// TwinCAT 3 PLC project PLC
// ProgramVersion: 3.1.4023.0
// libraries:
//   Tc2_MC2, * (Beckhoff Automation GmbH)
//   Tc2_PlcInterpolation, * (Beckhoff Automation GmbH)
//   Tc2_Standard, * (Beckhoff Automation GmbH)
//   Tc2_System, * (Beckhoff Automation GmbH)
//   Tc3_Module, * (Beckhoff Automation GmbH)
// project tree:
//   DUTs/ CASE_MODE.TcDUT, CASE_STATE.TcDUT, INIT_GVL.TcGVL, McOutputs.TcGVL, NCI_SingleEntry.TcDUT, PLCStruct.TcDUT, POS_REQ.TcDUT, POS_REQ_Resample.TcDUT, POS_RSP.TcDUT, POWER_GVL.TcGVL, RESET_GVL.TcGVL, TEST_STATE.TcDUT, VEL_REQ.TcDUT, VEL_RSP.TcDUT
//   / PlcTask.TcTTO
//   POUs/ AXIS.TcPOU, INIT.TcPOU, MAIN.TcPOU, Move_Vel.TcPOU, NCI_REF.TcPOU, POWER.TcPOU, PRG_MC_FeedTable.TcPOU, READ_POS.TcPOU, READ_VEL.TcPOU, RESET.TcPOU, SetPointGeneration.TcPOU, set_pos.TcPOU, TEST.TcPOU, TimeGet.TcPOU, WAIT.TcPOU

CONFIGURATION PLC
    RESOURCE PLC ON TwinCAT3
        TASK PlcTask(INTERVAL := T#50000us, PRIORITY := 20);
        PROGRAM MAIN WITH PlcTask : MAIN;
    END_RESOURCE
END_CONFIGURATION

// ---- DUTs/CASE_MODE.TcDUT

TYPE CASE_MODE :
(
	DEFAULT := 0,
	Set_PointGeneration,
	Set_Vel
);
END_TYPE

// ---- DUTs/CASE_STATE.TcDUT

TYPE CASE_STATE :
(
	ENUM_INIT_0 :=0,
	ENUM_POWER,
	ENUM_INIT,
	ENUM_SET_POSITION_GENERATION,
	ENUM_ERROR,
	ENUM_RESET
)INT;
END_TYPE

// ---- DUTs/NCI_SingleEntry.TcDUT
TYPE NCI_SingleEntry :
STRUCT
	SyncVelo:REAL;
	SyncAcc:REAL;
	fX:REAL;
	fY:REAL;
	fZ:REAL;
	
	fQ1:REAL;
	fQ2:REAL;
	
	fCenterX:REAL;
	fCenterY:REAL;
	fCenterZ:REAL;
	iPlane:REAL;
	
	Reserve1:UDINT;
	Reserve2:UDINT;
END_STRUCT
END_TYPE

// ---- DUTs/PLCStruct.TcDUT
TYPE PLCStruct :
STRUCT
	FLOAT1 :LREAL;
	FLOAT2 :LREAL;
	FLOAT3 :LREAL;
	FLOAT4 :LREAL;
(*
	intVal : INT;
	floatVal : REAL;
	boolVal : BOOL;
	*)
END_STRUCT
END_TYPE

// ---- DUTs/POS_REQ.TcDUT
TYPE POS_REQ :
STRUCT
	POS1: LREAL;
	POS2: LREAL;
	POS3: LREAL;
	POS4: LREAL;
	POS5: LREAL;
	POS6: LREAL;
END_STRUCT
END_TYPE

// ---- DUTs/POS_REQ_Resample.TcDUT
TYPE POS_REQ_Resample :
STRUCT
	POS_Resample: ARRAY[1..8,1..15] OF LREAL;
	(*POS1: LREAL;
	POS2: LREAL;
	POS3: LREAL;
	POS4: LREAL;
	POS5: LREAL;
	POS6: LREAL;*)

END_STRUCT
END_TYPE

// ---- DUTs/POS_RSP.TcDUT
TYPE POS_RSP :
STRUCT
	POS1: LREAL;
	POS2: LREAL;
	POS3: LREAL;
	POS4: LREAL;
	POS5: LREAL;
	POS6: LREAL;
END_STRUCT
END_TYPE

// ---- DUTs/TEST_STATE.TcDUT
TYPE TEST_STATE :
(
	TEST_0 :=0,
	TEST_1,
	TEST_2,
	TEST_3
)INT;
END_TYPE

// ---- DUTs/VEL_REQ.TcDUT
TYPE VEL_REQ :
STRUCT
	VEL5: LREAL;
	VEL6: LREAL;
END_STRUCT
END_TYPE

// ---- DUTs/VEL_RSP.TcDUT
TYPE VEL_RSP :
STRUCT
	VEL1: LREAL;
	VEL2: LREAL;
	VEL3: LREAL;
	VEL4: LREAL;
	VEL5: LREAL;
	VEL6: LREAL;
END_STRUCT
END_TYPE

// ---- DUTs/INIT_GVL.TcGVL

VAR_GLOBAL
	INIT_Execute1 : BOOL;
	INIT_Execute2 : BOOL;
	INIT_Execute3 : BOOL;
	INIT_Execute4 : BOOL;
	INIT_Execute5 : BOOL;
	INIT_Execute6 : BOOL;
END_VAR

// ---- DUTs/McOutputs.TcGVL

VAR_GLOBAL
	MC_Power_Outputs1: ST_McOutputs;
	MC_Power_Outputs2: ST_McOutputs;
	MC_Power_Outputs3: ST_McOutputs;
	MC_Power_Outputs4: ST_McOutputs;
	MC_Power_Outputs5: ST_McOutputs;
	MC_Power_Outputs6: ST_McOutputs;
END_VAR

// ---- DUTs/POWER_GVL.TcGVL

VAR_GLOBAL
	POWER_Enable1 : BOOL;
	POWER_Enable2 : BOOL;
	POWER_Enable3 : BOOL;
	POWER_Enable4 : BOOL;
	POWER_Enable5 : BOOL;
	POWER_Enable6 : BOOL;
END_VAR

// ---- DUTs/RESET_GVL.TcGVL

VAR_GLOBAL
	RESET_Execute1 : BOOL;
	RESET_Execute2 : BOOL;
	RESET_Execute3 : BOOL;
	RESET_Execute4 : BOOL;
	RESET_Execute5 : BOOL;
	RESET_Execute6 : BOOL;
END_VAR

// ---- POUs/MAIN.TcPOU
PROGRAM MAIN
VAR
	//BOOL1 AT %MX0.0 :BOOL;
	//INT2 AT %MD2 :INT;
	//FLOAT1 AT %MD6:REAL;
	//String1 : STRING;
	//Array1 : ARRAY[0..9] OF INT;
	//PLCVar:PLCStruct;
	//ArrayS:ARRAY[0..9] OF PLCStruct;
	//array2: ARRAY[1..50] OF LREAL:=[1,2,3,4,5,6,7,8,9,10,11,12,13,14,15,16,17,18,19,20,21,22,23,24,25,26,27,28,29,30,31,32,33,34,35,36,37,38,39,40,41,42,43,44,45,46,47,48,49,50];
	//TON1: TON;	
	//count: INT;
	//CTU1: CTU;

	CASE_MODE1 :CASE_MODE;
	FillFlag AT %MX0.0: BOOL;
	MoveDoneFlag AT %MX1.0: BOOL;
	Move_Stop_Flag AT %MX2.0: BOOL;
	Power_Flag AT %MX3.0: BOOL;
	Init_Flag AT %MX12.0: BOOL;
	NoPower_Flag AT %MX5.0: BOOL;
	Reset_Flag AT %MX6.0: BOOL;
	Continue_Flag AT %MX7.0: BOOL;
	Mode_Flag AT %MD8: INT;
	test1 AT %MX10.0: BOOL;
	test2 AT %MX11.0: BOOL;
	start_flag AT %MX9.0: BOOL;
	set_pos_flag AT %MX13.0: BOOL;
	err_flag AT %MX14.0: BOOL;
	Init_Done_flag AT %MX15.0: BOOL;
	MovePermit_Flag: BOOL;
	POS1_temp: LREAL;
	POS2_temp: LREAL;
	POS3_temp: LREAL;
	POS4_temp: LREAL;
	Done1Flag: LREAL;
	Done2Flag: LREAL;
	Done3Flag: LREAL;
	Done4Flag: LREAL;
	i: INT;
	x AT %MW2: INT;
	POS_REQ :POS_REQ;
	POS_RSP1 :POS_RSP;
	VEL_RSP1 :VEL_RSP;
	POS_REQ_Resample1:POS_REQ_Resample;	
	VEL_REQ1 :VEL_REQ;
	
	j: INT;
	m: INT;
	fbGetCurTaskIdx  : GETCURTASKINDEX;
    nLastExecTime       : UDINT;
	init_done_1: BOOL;
	init_done_2: BOOL;
	init_done_3: BOOL;
	init_done_4: BOOL;
	init_done_5: BOOL;
	init_done_6: BOOL;
END_VAR

//PRG_MC_FeedTable();
AXIS();
READ_POS();
READ_VEL();
//	IF AXIS.axis1.Status.Error AND AXIS.axis2.Status.Error AND AXIS.axis3.Status.Error AND AXIS.axis4.Status.Error THEN
//		start_flag:=0;
//	ELSE
//		start_flag:=1;
//	END_IF

		IF 	Move_Stop_Flag THEN
			MovePermit_Flag :=FALSE;
		END_IF
		IF Continue_Flag AND NOT err_flag THEN
			Move_Stop_Flag:= 0;
			MovePermit_Flag :=TRUE;
			Continue_Flag:= 0;
		END_IF
		IF Init_Flag AND NOT err_flag THEN
			POWER_Enable1:=TRUE; 
			POWER_Enable2:=TRUE;
			POWER_Enable3:=TRUE;
			POWER_Enable4:=TRUE;
			POWER();
			IF MC_Power_Outputs1.Done  AND MC_Power_Outputs2.Done AND MC_Power_Outputs3.Done AND MC_Power_Outputs4.Done THEN
				Power_Flag:= TRUE;
				INIT.MC_MoveAbsolute_1(Axis:=AXIS.Axis1,Execute:=TRUE,Position:=0,Velocity:=300);
				INIT.MC_MoveAbsolute_2(Axis:=AXIS.Axis2,Execute:=TRUE,Position:=0,Velocity:=300);
				INIT.MC_MoveAbsolute_3(Axis:=AXIS.Axis3,Execute:=TRUE,Position:=0,Velocity:=300);
				INIT.MC_MoveAbsolute_4(Axis:=AXIS.Axis4,Execute:=TRUE,Position:=0,Velocity:=300);
				IF NOT INIT.MC_MoveAbsolute_1.busy THEN
					init_done_1 := TRUE;
				END_IF
				IF NOT INIT.MC_MoveAbsolute_2.busy THEN
					init_done_2 := TRUE;
				END_IF
				IF NOT INIT.MC_MoveAbsolute_3.busy THEN
					init_done_3 := TRUE;
				END_IF
				IF NOT INIT.MC_MoveAbsolute_4.busy THEN
					init_done_4 := TRUE;
				END_IF
				IF init_done_1 AND init_done_2 AND init_done_3 AND init_done_4 THEN
					INIT.MC_MoveAbsolute_1(Axis:=AXIS.Axis1,Execute:=FALSE);
					INIT.MC_MoveAbsolute_2(Axis:=AXIS.Axis2,Execute:=FALSE);
					INIT.MC_MoveAbsolute_3(Axis:=AXIS.Axis3,Execute:=FALSE);
					INIT.MC_MoveAbsolute_4(Axis:=AXIS.Axis4,Execute:=FALSE);
					init_done_1 :=FALSE;
					init_done_2 :=FALSE;
					init_done_3 :=FALSE;
					init_done_4 :=FALSE;
					SetPointGeneration.MC_ExtSetPointGenEnable1(Axis:=AXIS.Axis1,Execute:=FALSE);	
					SetPointGeneration.MC_ExtSetPointGenEnable2(Axis:=AXIS.Axis2,Execute:=FALSE);
					SetPointGeneration.MC_ExtSetPointGenEnable3(Axis:=AXIS.Axis3,Execute:=FALSE);
					SetPointGeneration.MC_ExtSetPointGenEnable4(Axis:=AXIS.Axis4,Execute:=FALSE);
					SetPointGeneration.MC_ExtSetPointGenDisable1(Axis:=AXIS.Axis1,Execute:=FALSE);	
					SetPointGeneration.MC_ExtSetPointGenDisable2(Axis:=AXIS.Axis2,Execute:=FALSE);
					SetPointGeneration.MC_ExtSetPointGenDisable3(Axis:=AXIS.Axis3,Execute:=FALSE);
					SetPointGeneration.MC_ExtSetPointGenDisable4(Axis:=AXIS.Axis4,Execute:=FALSE);
					Init_Flag:= 0;
					Power_Flag:= 0;
					MovePermit_Flag:= 1;
					Init_Done_flag:=1;
				END_IF
			END_IF
			IF AXIS.axis1.Status.Error AND AXIS.axis2.Status.Error AND AXIS.axis3.Status.Error AND AXIS.axis4.Status.Error THEN
				err_flag:=1;
			END_IF					
		END_IF
		
		IF set_pos_flag THEN
			set_pos.MC_SetPosition1(axis:=axis.Axis1,execute:=FALSE,position:=0);
			set_pos.MC_SetPosition2(axis:=axis.Axis2,execute:=FALSE,position:=0);
			set_pos.MC_SetPosition3(axis:=axis.Axis3,execute:=FALSE,position:=0);
			set_pos.MC_SetPosition4(axis:=axis.Axis4,execute:=FALSE,position:=0);
			set_pos.MC_SetPosition1(axis:=axis.Axis1,execute:=TRUE,position:=0);
			set_pos.MC_SetPosition2(axis:=axis.Axis2,execute:=TRUE,position:=0);
			set_pos.MC_SetPosition3(axis:=axis.Axis3,execute:=TRUE,position:=0);
			set_pos.MC_SetPosition4(axis:=axis.Axis4,execute:=TRUE,position:=0);
			set_pos_flag:=0;
		END_IF
		
		IF Reset_Flag THEN
			SetPointGeneration.MC_ExtSetPointGenDisable1(Axis:=AXIS.Axis1,Execute:=TRUE);	
			SetPointGeneration.MC_ExtSetPointGenDisable2(Axis:=AXIS.Axis2,Execute:=TRUE);
			SetPointGeneration.MC_ExtSetPointGenDisable3(Axis:=AXIS.Axis3,Execute:=TRUE);
			SetPointGeneration.MC_ExtSetPointGenDisable4(Axis:=AXIS.Axis4,Execute:=TRUE);
			INIT.MC_MoveAbsolute_1(Axis:=AXIS.Axis1,Execute:=FALSE);
			INIT.MC_MoveAbsolute_2(Axis:=AXIS.Axis2,Execute:=FALSE);
			INIT.MC_MoveAbsolute_3(Axis:=AXIS.Axis3,Execute:=FALSE);
			INIT.MC_MoveAbsolute_4(Axis:=AXIS.Axis4,Execute:=FALSE);
			Init_Flag :=FALSE;
			POWER_Enable1:=FALSE;
			POWER_Enable2:=FALSE;
			POWER_Enable3:=FALSE;
			POWER_Enable4:=FALSE;
			POWER();
			Power_Flag :=0;
			RESET.MC_Reset1(Axis:=AXIS.Axis1,Execute:=TRUE);
			RESET.MC_Reset2(Axis:=AXIS.Axis2,Execute:=TRUE);
			RESET.MC_Reset3(Axis:=AXIS.Axis3,Execute:=TRUE);
			RESET.MC_Reset4(Axis:=AXIS.Axis4,Execute:=TRUE);
			RESET.MC_Reset1(Axis:=AXIS.Axis1,Execute:=FALSE);
			RESET.MC_Reset2(Axis:=AXIS.Axis2,Execute:=FALSE);
			RESET.MC_Reset3(Axis:=AXIS.Axis3,Execute:=FALSE);
			RESET.MC_Reset4(Axis:=AXIS.Axis4,Execute:=FALSE);
			Reset_Flag:= 0;
			Init_Done_flag:=0;
			NoPower_Flag:= 0;
			Move_Stop_Flag:= 0;
			MovePermit_Flag:= 0;
			start_flag:=0;
		END_IF
		IF NoPower_Flag AND NOT err_flag THEN
			MovePermit_Flag:= 0;
			Init_Flag:= 0;
			NoPower_Flag:= FALSE;
			POWER_Enable1:=FALSE;
			POWER_Enable2:=FALSE;
			POWER_Enable3:=FALSE;
			POWER_Enable4:=FALSE;
			POWER();
	//IF SetPointGeneration.MC_Power_1_Outputs.Done AND SetPointGeneration.MC_Power_2_Outputs.Done AND SetPointGeneration.MC_Power_3_Outputs.Done AND SetPointGeneration.MC_Power_4_Outputs.Done THEN
		
	//END_IF	
		END_IF
		IF MovePermit_Flag AND NOT err_flag THEN
			FillFlag:= FALSE;
			IF MOve_Stop_Flag THEN
				;
			ELSE
				i:= i+1;
			END_IF

			x:= i MOD 15;
	
			POS_RSP1.POS1:= AXIS.Axis1.NcToPlc.actPos;
			POS_RSP1.POS2:= AXIS.Axis2.NcToPlc.actPos;
			POS_RSP1.POS3:= AXIS.Axis3.NcToPlc.actPos;
			POS_RSP1.POS4:= AXIS.Axis4.NcToPlc.actPos;
			VEL_RSP1.VEL1:= AXIS.Axis1.NcToPlc.actVelo;
			VEL_RSP1.VEL2:= AXIS.Axis2.NcToPlc.actVelo;
			VEL_RSP1.VEL3:= AXIS.Axis3.NcToPlc.actVelo;
			VEL_RSP1.VEL4:= AXIS.Axis4.NcToPlc.actVelo;
			Done1Flag:=AXIS.Axis1.NcToPlc.actPos-POS1_temp;
			Done2Flag:=AXIS.Axis2.NcToPlc.actPos-POS2_temp;
			Done3Flag:=AXIS.Axis3.NcToPlc.actPos-POS3_temp;
			Done4Flag:=AXIS.Axis4.NcToPlc.actPos-POS4_temp;

			IF MOve_Stop_Flag = 0 AND ABS(Done1Flag)<1E-3 AND ABS(Done2Flag)<1E-3 AND ABS(Done3Flag)<1E-3 AND ABS(Done4Flag)<1E-3 THEN
				MoveDoneFlag:= 1;
			ELSE
				MoveDoneFlag:= 0;
			END_IF
	
			POS_REQ.POS1:= -POS_REQ_Resample1.POS_Resample[3,x+1];
			POS_REQ.POS2:= -POS_REQ_Resample1.POS_Resample[4,x+1];
			POS_REQ.POS3:= -POS_REQ_Resample1.POS_Resample[1,x+1];
			POS_REQ.POS4:= -POS_REQ_Resample1.POS_Resample[2,x+1];
			IF POS_REQ_Resample1.POS_Resample[7,x] = 1 THEN
				POS1_temp:= POS_REQ.POS1;
			END_IF
			IF POS_REQ_Resample1.POS_Resample[8,x] = 1 THEN
				POS2_temp:= POS_REQ.POS2;
			END_IF
			IF POS_REQ_Resample1.POS_Resample[5,x] = 1 THEN
				POS3_temp:= POS_REQ.POS3;
			END_IF
			IF POS_REQ_Resample1.POS_Resample[6,x] = 1 THEN
				POS4_temp:= POS_REQ.POS4;
			END_IF

		SetPointGeneration.MC_ExtSetPointGenEnable1(Axis:=AXIS.Axis1,Execute:=TRUE,Position:=POS_REQ.POS1);	
		SetPointGeneration.MC_ExtSetPointGenEnable2(Axis:=AXIS.Axis2,Execute:=TRUE,Position:=POS_REQ.POS2);
		SetPointGeneration.MC_ExtSetPointGenEnable3(Axis:=AXIS.Axis3,Execute:=TRUE,Position:=POS_REQ.POS3);
		SetPointGeneration.MC_ExtSetPointGenEnable4(Axis:=AXIS.Axis4,Execute:=TRUE,Position:=POS_REQ.POS4);
		IF SetPointGeneration.MC_ExtSetPointGenEnable1.Enabled AND  SetPointGeneration.MC_ExtSetPointGenEnable2.Enabled AND  SetPointGeneration.MC_ExtSetPointGenEnable3.Enabled AND  SetPointGeneration.MC_ExtSetPointGenEnable4.Enabled THEN
			MC_ExtSetPointGenFeed(
				Position:= MAIN.POS_REQ.POS1, 		
				Velocity:= 1, 
				Acceleration:=1 , 
				Direction:= 1,
				Axis:= AXIS.Axis1);	
			MC_ExtSetPointGenFeed(
				Position:= MAIN.POS_REQ.POS2, 		
				Velocity:= 1, 
				Acceleration:=1 , 
				Direction:= 1,
				Axis:= AXIS.Axis2);	
			MC_ExtSetPointGenFeed(
				Position:= MAIN.POS_REQ.POS3, 		
				Velocity:= 1, 
				Acceleration:=1 , 
				Direction:= 1,
				Axis:= AXIS.Axis3);	
			MC_ExtSetPointGenFeed(
				Position:= MAIN.POS_REQ.POS4, 		
				Velocity:= 1, 
				Acceleration:=1 , 
				Direction:= 1,
				Axis:= AXIS.Axis4);		
				
		END_IF
		IF AXIS.axis1.Status.Error AND AXIS.axis2.Status.Error AND AXIS.axis3.Status.Error AND AXIS.axis4.Status.Error THEN
			err_flag := 1;
		END_IF
	
			IF x = 14 AND MOve_Stop_Flag = 0 THEN
				FillFlag:= TRUE;
		(*FOR m:= 1 TO 15 DO
			POS_REQ_Resample1.POS_Resample[1,m]:=15*j+m;
		END_FOR
		j:= j+1;*)
			END_IF
	
		END_IF
		IF err_flag THEN
			Reset_Flag:=1;
			IF NOT AXIS.axis1.Status.Error AND NOT AXIS.axis2.Status.Error AND NOT AXIS.axis3.Status.Error AND NOT AXIS.axis4.Status.Error THEN
				err_flag := 0;
			END_IF
		END_IF
		
fbGetCurTaskIdx();
nLastExecTime := _TaskInfo[fbGetCurTaskIdx.index].LastExecTime;

END_PROGRAM

// ---- POUs/AXIS.TcPOU
PROGRAM AXIS
VAR
	Axis1: AXIS_REF;
	Axis2: AXIS_REF;
	Axis3: AXIS_REF;
	Axis4: AXIS_REF;
	Axis5: AXIS_REF;
	Axis6: AXIS_REF;
END_VAR

Axis1(
	PlcToNc:= , 
	NcToPlc=> , 
	ADS=> , 
	Status=> , 
	DriveAddress:= );
	
Axis2(
	PlcToNc:= , 
	NcToPlc=> , 
	ADS=> , 
	Status=> , 
	DriveAddress:= );
	
Axis3(
	PlcToNc:= , 
	NcToPlc=> , 
	ADS=> , 
	Status=> , 
	DriveAddress:= );
	
Axis4(
	PlcToNc:= , 
	NcToPlc=> , 
	ADS=> , 
	Status=> , 
	DriveAddress:= );

Axis5(
	PlcToNc:= , 
	NcToPlc=> , 
	ADS=> , 
	Status=> , 
	DriveAddress:= );
	
Axis6(
	PlcToNc:= , 
	NcToPlc=> , 
	ADS=> , 
	Status=> , 
	DriveAddress:= );

END_PROGRAM

// ---- POUs/READ_POS.TcPOU
PROGRAM READ_POS
VAR
	MC_ReadActualPosition1 : MC_ReadActualPosition;
	MC_ReadActualPosition2 : MC_ReadActualPosition;
	MC_ReadActualPosition3 : MC_ReadActualPosition;
	MC_ReadActualPosition4 : MC_ReadActualPosition;
END_VAR

MC_ReadActualPosition1(
	Axis:= AXIS.Axis1, 
	Enable:= , 
	Valid=> , 
	Busy=> , 
	Error=> , 
	ErrorID=> , 
	Position=> );
	
MC_ReadActualPosition2(
	Axis:= AXIS.Axis2, 
	Enable:= , 
	Valid=> , 
	Busy=> , 
	Error=> , 
	ErrorID=> , 
	Position=> );
	
MC_ReadActualPosition3(
	Axis:= AXIS.Axis3, 
	Enable:= , 
	Valid=> , 
	Busy=> , 
	Error=> , 
	ErrorID=> , 
	Position=> );
	
MC_ReadActualPosition4(
	Axis:= AXIS.Axis4, 
	Enable:= , 
	Valid=> , 
	Busy=> , 
	Error=> , 
	ErrorID=> , 
	Position=> );

END_PROGRAM

// ---- POUs/READ_VEL.TcPOU
PROGRAM READ_VEL
VAR
	MC_ReadActualVelocity1 : MC_ReadActualVelocity;
	MC_ReadActualVelocity2 : MC_ReadActualVelocity;
	MC_ReadActualVelocity3 : MC_ReadActualVelocity;
	MC_ReadActualVelocity4 : MC_ReadActualVelocity;
END_VAR

MC_ReadActualVelocity1(
	Axis:= AXIS.Axis1, 
	Enable:= , 
	Valid=> , 
	Busy=> , 
	Error=> , 
	ErrorID=> , 
	ActualVelocity=> );
	
MC_ReadActualVelocity2(
	Axis:= AXIS.Axis2, 
	Enable:= , 
	Valid=> , 
	Busy=> , 
	Error=> , 
	ErrorID=> , 
	ActualVelocity=> );
	
MC_ReadActualVelocity3(
	Axis:= AXIS.Axis3, 
	Enable:= , 
	Valid=> , 
	Busy=> , 
	Error=> , 
	ErrorID=> , 
	ActualVelocity=> );
	
MC_ReadActualVelocity4(
	Axis:= AXIS.Axis4, 
	Enable:= , 
	Valid=> , 
	Busy=> , 
	Error=> , 
	ErrorID=> , 
	ActualVelocity=> );

END_PROGRAM

// ---- POUs/POWER.TcPOU
PROGRAM POWER
VAR
	MC_Power_1: MC_Power;
	MC_Power_2: MC_Power;
	MC_Power_3: MC_Power;
	MC_Power_4: MC_Power;
	MC_Power_5: MC_Power;
	MC_Power_6: MC_Power;
	
END_VAR

MC_Power_1(
	Axis:= AXIS.Axis1, 
	Enable:= POWER_Enable1, 
	Enable_Positive:= POWER_Enable1, 
	Enable_Negative:= POWER_Enable1, 
	Override:= , 
	BufferMode:= , 
	Options:= , 
	Status=> MC_Power_Outputs1.Done, 
	Busy=> MC_Power_Outputs1.Busy, 
	Active=> MC_Power_Outputs1.Active, 
	Error=> MC_Power_Outputs1.Error, 
	ErrorID=> MC_Power_Outputs1.ErrorID);
	
MC_Power_2(
	Axis:= AXIS.Axis2, 
	Enable:= POWER_Enable2, 
	Enable_Positive:= POWER_Enable2, 
	Enable_Negative:= POWER_Enable2, 
	Override:= , 
	BufferMode:= , 
	Options:= , 
	Status=> MC_Power_Outputs2.Done, 
	Busy=> MC_Power_Outputs2.Busy, 
	Active=> MC_Power_Outputs2.Active, 
	Error=> MC_Power_Outputs2.Error, 
	ErrorID=> MC_Power_Outputs2.ErrorID);
	
MC_Power_3(
	Axis:= AXIS.Axis3, 
	Enable:= POWER_Enable3, 
	Enable_Positive:= POWER_Enable3, 
	Enable_Negative:= POWER_Enable3, 
	Override:= , 
	BufferMode:= , 
	Options:= , 
	Status=> MC_Power_Outputs3.Done, 
	Busy=> MC_Power_Outputs3.Busy, 
	Active=> MC_Power_Outputs3.Active, 
	Error=> MC_Power_Outputs3.Error, 
	ErrorID=> MC_Power_Outputs3.ErrorID);
	
MC_Power_4(
	Axis:= AXIS.Axis4, 
	Enable:= POWER_Enable4, 
	Enable_Positive:= POWER_Enable4, 
	Enable_Negative:= POWER_Enable4, 
	Override:= , 
	BufferMode:= , 
	Options:= , 
	Status=> MC_Power_Outputs4.Done, 
	Busy=> MC_Power_Outputs4.Busy, 
	Active=> MC_Power_Outputs4.Active, 
	Error=> MC_Power_Outputs4.Error, 
	ErrorID=> MC_Power_Outputs4.ErrorID);
	
MC_Power_5(
	Axis:= AXIS.Axis5, 
	Enable:= POWER_Enable5, 
	Enable_Positive:= POWER_Enable5, 
	Enable_Negative:= POWER_Enable5, 
	Override:= , 
	BufferMode:= , 
	Options:= , 
	Status=> MC_Power_Outputs5.Done, 
	Busy=> MC_Power_Outputs5.Busy, 
	Active=> MC_Power_Outputs5.Active, 
	Error=> MC_Power_Outputs5.Error, 
	ErrorID=> MC_Power_Outputs5.ErrorID);
	
MC_Power_6(
	Axis:= AXIS.Axis6, 
	Enable:= POWER_Enable6, 
	Enable_Positive:= POWER_Enable6, 
	Enable_Negative:= POWER_Enable6, 
	Override:= , 
	BufferMode:= , 
	Options:= , 
	Status=> MC_Power_Outputs6.Done, 
	Busy=> MC_Power_Outputs6.Busy, 
	Active=> MC_Power_Outputs6.Active, 
	Error=> MC_Power_Outputs6.Error, 
	ErrorID=> MC_Power_Outputs6.ErrorID);

END_PROGRAM

// ---- POUs/INIT.TcPOU
PROGRAM INIT
VAR
	MC_MoveAbsolute_1 : MC_MoveAbsolute;
	MC_MoveAbsolute_2 : MC_MoveAbsolute;
	MC_MoveAbsolute_3 : MC_MoveAbsolute;
	MC_MoveAbsolute_4 : MC_MoveAbsolute;
	MC_MoveAbsolute_5 : MC_MoveAbsolute;
	MC_MoveAbsolute_6 : MC_MoveAbsolute;
END_VAR

MC_MoveAbsolute_1(
	Axis:= AXIS.Axis1, 
	Execute:= INIT_Execute1, 
	Position:= , 
	Velocity:= , 
	Acceleration:= , 
	Deceleration:= , 
	Jerk:= , 
	BufferMode:= , 
	Options:= , 
	Done=> , 
	Busy=> , 
	Active=> , 
	CommandAborted=> , 
	Error=> , 
	ErrorID=> );
	
MC_MoveAbsolute_2(
	Axis:= AXIS.Axis2, 
	Execute:= INIT_Execute2, 
	Position:= , 
	Velocity:= , 
	Acceleration:= , 
	Deceleration:= , 
	Jerk:= , 
	BufferMode:= , 
	Options:= , 
	Done=> , 
	Busy=> , 
	Active=> , 
	CommandAborted=> , 
	Error=> , 
	ErrorID=> );
	
MC_MoveAbsolute_3(
	Axis:= AXIS.Axis3, 
	Execute:= INIT_Execute3, 
	Position:= , 
	Velocity:= , 
	Acceleration:= , 
	Deceleration:= , 
	Jerk:= , 
	BufferMode:= , 
	Options:= , 
	Done=> , 
	Busy=> , 
	Active=> , 
	CommandAborted=> , 
	Error=> , 
	ErrorID=> );
	
MC_MoveAbsolute_4(
	Axis:= AXIS.Axis4, 
	Execute:= INIT_Execute4, 
	Position:= , 
	Velocity:= , 
	Acceleration:= , 
	Deceleration:= , 
	Jerk:= , 
	BufferMode:= , 
	Options:= , 
	Done=> , 
	Busy=> , 
	Active=> , 
	CommandAborted=> , 
	Error=> , 
	ErrorID=> );
	
MC_MoveAbsolute_5(
	Axis:= AXIS.Axis5, 
	Execute:= INIT_Execute5, 
	Position:= , 
	Velocity:= , 
	Acceleration:= , 
	Deceleration:= , 
	Jerk:= , 
	BufferMode:= , 
	Options:= , 
	Done=> , 
	Busy=> , 
	Active=> , 
	CommandAborted=> , 
	Error=> , 
	ErrorID=> );
	
MC_MoveAbsolute_6(
	Axis:= AXIS.Axis6, 
	Execute:= INIT_Execute6, 
	Position:= , 
	Velocity:= , 
	Acceleration:= , 
	Deceleration:= , 
	Jerk:= , 
	BufferMode:= , 
	Options:= , 
	Done=> , 
	Busy=> , 
	Active=> , 
	CommandAborted=> , 
	Error=> , 
	ErrorID=> );

END_PROGRAM

// ---- POUs/SetPointGeneration.TcPOU
PROGRAM SetPointGeneration
VAR
	
	CASE_STATE1: CASE_STATE;
	
	MC_ExtSetPointGenEnable1: MC_ExtSetPointGenEnable;
	MC_ExtSetPointGenEnable2: MC_ExtSetPointGenEnable;
	MC_ExtSetPointGenEnable3: MC_ExtSetPointGenEnable;
	MC_ExtSetPointGenEnable4: MC_ExtSetPointGenEnable;
	
	MC_ExtSetPointGenDisable1: MC_ExtSetPointGenDisable;
	MC_ExtSetPointGenDisable2: MC_ExtSetPointGenDisable;
	MC_ExtSetPointGenDisable3: MC_ExtSetPointGenDisable;
	MC_ExtSetPointGenDisable4: MC_ExtSetPointGenDisable;
	
END_VAR

AXIS();



MC_ExtSetPointGenEnable1(
	Axis:= AXIS.Axis1, 
	Execute:= , 
	Position:= , 
	PositionType:= , 
	Done=> , 
	Busy=> , 
	Error=> , 
	ErrorID=> , 
	Enabled=> );
	
MC_ExtSetPointGenEnable2(
	Axis:= AXIS.Axis2, 
	Execute:= , 
	Position:= , 
	PositionType:= , 
	Done=> , 
	Busy=> , 
	Error=> , 
	ErrorID=> , 
	Enabled=> );
	
MC_ExtSetPointGenEnable3(
	Axis:= AXIS.Axis3, 
	Execute:= , 
	Position:= , 
	PositionType:= , 
	Done=> , 
	Busy=> , 
	Error=> , 
	ErrorID=> , 
	Enabled=> );
	
MC_ExtSetPointGenEnable4(
	Axis:= AXIS.Axis4, 
	Execute:= , 
	Position:= , 
	PositionType:= , 
	Done=> , 
	Busy=> , 
	Error=> , 
	ErrorID=> , 
	Enabled=> );
	
	MC_ExtSetPointGenDisable1(
	Axis:= AXIS.Axis1, 
	Execute:= , 
	Done=> , 
	Busy=> , 
	Error=> , 
	ErrorID=> , 
	Enabled=> );
	
	MC_ExtSetPointGenDisable2(
	Axis:= AXIS.Axis2, 
	Execute:= , 
	Done=> , 
	Busy=> , 
	Error=> , 
	ErrorID=> , 
	Enabled=> );
	
	MC_ExtSetPointGenDisable3(
	Axis:= AXIS.Axis3, 
	Execute:= , 
	Done=> , 
	Busy=> , 
	Error=> , 
	ErrorID=> , 
	Enabled=> );
	
	MC_ExtSetPointGenDisable4(
	Axis:= AXIS.Axis4, 
	Execute:= , 
	Done=> , 
	Busy=> , 
	Error=> , 
	ErrorID=> , 
	Enabled=> );

	
		
	
//	ENUM_ERROR:
//		MC_ExtSetPointGenEnable1.Execute:=FALSE;
//		MC_ExtSetPointGenEnable2.Execute:=FALSE;
//		MC_ExtSetPointGenEnable3.Execute:=FALSE;
//		MC_ExtSetPointGenEnable4.Execute:=FALSE;
//		MC_ExtSetPointGenDisable1.Execute := MC_ExtSetPointGenEnable1.Enabled;	
//		MC_ExtSetPointGenDisable2.Execute := MC_ExtSetPointGenEnable2.Enabled;
//		MC_ExtSetPointGenDisable3.Execute := MC_ExtSetPointGenEnable3.Enabled;
//		MC_ExtSetPointGenDisable4.Execute := MC_ExtSetPointGenEnable4.Enabled;	
//		IF NOT AXIS.axis1.Status.Coupled AND AXIS.axis2.Status.Coupled AND AXIS.axis3.Status.Coupled AND AXIS.axis4.Status.Coupled THEN
//			IF AXIS.axis1.Status.Error AND AXIS.axis2.Status.Error AND AXIS.axis3.Status.Error AND AXIS.axis4.Status.Error THEN
//				CASE_STATE1 := ENUM_RESET;	
//			ELSE
//				CASE_STATE1 := ENUM_INIT_0;
//			END_IF
//		END_IF
	
//	ENUM_RESET:
//		RESET_Execute1 := TRUE;
//		RESET_Execute2 := TRUE;
//		RESET_Execute3 := TRUE;
//		RESET_Execute4 := TRUE;
//		RESET();
//		MC_ExtSetPointGenDisable1.Execute:=FALSE;
//		MC_ExtSetPointGenDisable2.Execute:=FALSE;
//		MC_ExtSetPointGenDisable3.Execute:=FALSE;
//		MC_ExtSetPointGenDisable4.Execute:=FALSE;		
//			IF RESET.MC_Reset1.Done AND RESET.MC_Reset2.Done AND RESET.MC_Reset3.Done AND RESET.MC_Reset4.Done THEN
//				CASE_STATE1 := ENUM_INIT_0;
//			ELSIF RESET.MC_Reset1.Error AND RESET.MC_Reset2.Error AND RESET.MC_Reset3.Error AND RESET.MC_Reset4.Error THEN
//				CASE_STATE1 := ENUM_INIT_0; 
//			END_IF

END_PROGRAM

// ---- POUs/set_pos.TcPOU
PROGRAM set_pos
VAR
	MC_SetPosition1: MC_SetPosition;
	MC_SetPosition2: MC_SetPosition;
	MC_SetPosition3: MC_SetPosition;
	MC_SetPosition4: MC_SetPosition;
	MC_SetPosition5: MC_SetPosition;
	MC_SetPosition6: MC_SetPosition;
END_VAR

MC_SetPosition1(
	Axis:= axis.Axis1, 
	Execute:= , 
	Position:= , 
	Mode:= , 
	Options:= , 
	Done=> , 
	Busy=> , 
	Error=> , 
	ErrorID=> );

MC_SetPosition2(
	Axis:= axis.Axis2, 
	Execute:= , 
	Position:= , 
	Mode:= , 
	Options:= , 
	Done=> , 
	Busy=> , 
	Error=> , 
	ErrorID=> );
	
MC_SetPosition3(
	Axis:= axis.Axis3, 
	Execute:= , 
	Position:= , 
	Mode:= , 
	Options:= , 
	Done=> , 
	Busy=> , 
	Error=> , 
	ErrorID=> );

MC_SetPosition4(
	Axis:= axis.Axis4, 
	Execute:= , 
	Position:= , 
	Mode:= , 
	Options:= , 
	Done=> , 
	Busy=> , 
	Error=> , 
	ErrorID=> );
	
MC_SetPosition5(
	Axis:= axis.Axis5, 
	Execute:= , 
	Position:= , 
	Mode:= , 
	Options:= , 
	Done=> , 
	Busy=> , 
	Error=> , 
	ErrorID=> );

MC_SetPosition6(
	Axis:= axis.Axis6, 
	Execute:= , 
	Position:= , 
	Mode:= , 
	Options:= , 
	Done=> , 
	Busy=> , 
	Error=> , 
	ErrorID=> );

END_PROGRAM

// ---- POUs/RESET.TcPOU
PROGRAM RESET
VAR
	MC_Reset1 : MC_Reset;
	MC_Reset2 : MC_Reset;
	MC_Reset3 : MC_Reset;
	MC_Reset4 : MC_Reset;
	MC_Reset5 : MC_Reset;
	MC_Reset6 : MC_Reset;
END_VAR

MC_Reset1(
	Axis:= AXIS.Axis1, 
	Execute:= RESET_Execute1, 
	Done=> , 
	Busy=> , 
	Error=> , 
	ErrorID=> );
	
	MC_Reset2(
	Axis:= AXIS.Axis2, 
	Execute:= RESET_Execute2, 
	Done=> , 
	Busy=> , 
	Error=> , 
	ErrorID=> );
	
	MC_Reset3(
	Axis:= AXIS.Axis3, 
	Execute:= RESET_Execute3, 
	Done=> , 
	Busy=> , 
	Error=> , 
	ErrorID=> );
	
	MC_Reset4(
	Axis:= AXIS.Axis4, 
	Execute:= RESET_Execute4, 
	Done=> , 
	Busy=> , 
	Error=> , 
	ErrorID=> );
	
	MC_Reset5(
	Axis:= AXIS.Axis5, 
	Execute:= RESET_Execute5, 
	Done=> , 
	Busy=> , 
	Error=> , 
	ErrorID=> );
	
	MC_Reset6(
	Axis:= AXIS.Axis6, 
	Execute:= RESET_Execute6, 
	Done=> , 
	Busy=> , 
	Error=> , 
	ErrorID=> );

END_PROGRAM

// ---- POUs/Move_Vel.TcPOU
PROGRAM Move_Vel
VAR
	MC_MoveVelocity5: MC_MoveVelocity;
	MC_MoveVelocity6: MC_MoveVelocity;
END_VAR


AXIS();

MC_MoveVelocity5(
	Axis:= AXIS.Axis5, 
	Execute:= , 
	Velocity:= MAIN.VEL_REQ1.VEL5, 
	Acceleration:= , 
	Deceleration:= , 
	Jerk:= , 
	Direction:= , 
	BufferMode:= , 
	Options:= , 
	InVelocity=> , 
	Busy=> , 
	Active=> , 
	CommandAborted=> , 
	Error=> , 
	ErrorID=> );
MC_MoveVelocity6(
	Axis:= AXIS.Axis6, 
	Execute:= , 
	Velocity:= MAIN.VEL_REQ1.VEL6, 
	Acceleration:= , 
	Deceleration:= , 
	Jerk:= , 
	Direction:= , 
	BufferMode:= , 
	Options:= , 
	InVelocity=> , 
	Busy=> , 
	Active=> , 
	CommandAborted=> , 
	Error=> , 
	ErrorID=> );

END_PROGRAM

// ---- POUs/NCI_REF.TcPOU
FUNCTION_BLOCK NCI_REF
VAR_INPUT
END_VAR
VAR_OUTPUT
END_VAR
VAR
	PlcToNci AT %Q* : PLCTONC_NCICHANNEL_REF;
	NciToPlc AT %I* : NcToPlc_NciChannel_Ref;
END_VAR

END_FUNCTION_BLOCK

// ---- POUs/PRG_MC_FeedTable.TcPOU
PROGRAM PRG_MC_FeedTable
VAR
	(*NCI 通道的 Axis 和 Channel ，与 TwinCAT NC 的接口变量*)
AxisX :AXIS_REF;
AxisY :AXIS_REF;
ItpChannel :NCI_REF;
(*基本动作功能块：通道组合，通道解散，装载 G 代码文件，启动停止，复位*)
CfgBuildExt3DGroup : CfgBuildExt3DGroup;
fbClearGrp :CfgReconfigGroup; 
fbItpStartStop :ItpStartStop;
fbItpReset :ItpResetEx2;
TblPrep : FB_NciFeedTablePreparation;
NCI_Entry : NCI_SingleEntry;
(*自定义结构体：准备赋给待填充指令 GeoCircleCIP 和 GeoLine 的数据*)
GeoCircleCIP : ST_NciGeoCircleCIP;
(*待填充到 Table 的圆弧插补指令*)
GeoLine : ST_NciGeoLine;
(*待填充到 Table 的直线插补指令*)
NciFeedTable :FB_NciFeedTable;
Table : ST_NciFeedGroupTable;
(*插补通道要执行的插补指令序列*)
TableDisplayIndex : UDINT := 1;
(*插补指令在 Table 中的索引号*)
rOverride :LREAL := 100;
(*插补运动的倍率*)
(*通道 ID 和轴组 ID*)
GroupID : UDINT;
ChannelID : UDINT;
(*仅在数据准备的上升沿，才把 Entry 中的数据填充到 Table*)
bTablePrepare :BOOL;
fbRTrigTablePrepare :R_TRIG;
END_VAR

(*引用 4 个 Action ，实现不同的功能*)
M_PTP(); (*轴使能*)
M_BasicFB(); (*NCI 通道控制*)
M_UpdateStatus(); (*NCI 通道状态刷新*)
M_GoPLine(); (*数据填充*)

(*准备手动控制 NC 通道的触发命令*)
rOverride;
CfgBuildExt3DGroup.bExecute;
fbClearGrp.bExecute;
fbItpReset.bExecute;
NCI_Entry.fX;
NCI_Entry.fY;
NCI_Entry.SyncVelo;
bTablePrepare;
TblPrep.bResetTable;
NciFeedTable.bExecute;

ACTION M_BasicFB:
CfgBuildExt3DGroup(
bExecute:= ,
nGroupId:=GroupID ,
nXAxisId:=AxisX.NcToPlc.AxisId ,
nYAxisId:=AxisY.NcToPlc.AxisId ,
nZAxisId:=,
nQ1AxisId:=,
nQ2AxisId:=,
tTimeOut:=T#500ms ,
bBusy=> ,
bErr=> ,
nErrId=> );

fbClearGrp(
bExecute:= ,
nGroupId:= GroupID ,
tTimeOut:= T#500MS);

fbItpStartStop(
bStart:= ,
bStop:= ,
nChnId:=ChannelID,
tTimeOut:=T#500MS ,
bBusy=> ,
bErr=> ,
nErrId=> );

fbItpReset(
bExecute:= ,
tTimeOut:= T#500MS,
sNciToPlc:= ItpChannel.NciToPlc,
bBusy=> ,
bErr=> ,
nErrId=> );

TblPrep(
nEntryType := ,
pEntry := ,
bResetTable:= ,
stFeedGroupTable:= Table,
nFilledRows=> ,
bError => ,
nErrorId => );

NciFeedTable(
bExecute:= ,
bReset:= ,
bLogFeederEntries:= FALSE ,
stFeedGroupTable:= Table,
stNciToPlc:=ItpChannel.NciToPlc );
END_ACTION

ACTION M_GoPLine:
fbRTrigTablePrepare(CLK:=bTablePrepare , Q=> );
IF NOT fbRTrigTablePrepare.Q THEN RETURN; END_IF (* 仅当上升沿才往Table 里填一条数据*)
IF NCI_Entry.SyncVelo >0.001 THEN
IF NCI_Entry.iPlane>0 THEN (*Circle*)
GeoCircleCIP.fEndPosX:= REAL_TO_LREAL(NCI_Entry.fX);
GeoCircleCIP.fEndPosY:=  REAL_TO_LREAL(NCI_Entry.fY);
GeoCircleCIP.fCIPPosX:=  REAL_TO_LREAL(NCI_Entry.fCenterX);
GeoCircleCIP.fCIPPosY:=  REAL_TO_LREAL(NCI_Entry.fCenterY);
GeoCircleCIP.fVelo:=  REAL_TO_LREAL(NCI_Entry.SyncVelo);
TableDisplayIndex:=  TableDisplayIndex+1;
GeoLine.nDisplayIndex := TableDisplayIndex;
TblPrep.nEntryType:=  GeoCircleCIP.nEntryType;
TblPrep.pEntry:=  ADR(GeoCircleCIP);
TblPrep.bResetTable:=  FALSE;
ELSE (*Line*)
GeoLine.fEndPosX:=  REAL_TO_LREAL(NCI_Entry.fX);
GeoLine.fEndPosY:=  REAL_TO_LREAL(NCI_Entry.fY);
GeoLine.fEndPosZ:=  REAL_TO_LREAL(NCI_Entry.fZ);
GeoLine.fEndPosQ1:=  REAL_TO_LREAL(NCI_Entry.fQ1);
GeoLine.fEndPosQ2:=  REAL_TO_LREAL(NCI_Entry.fQ2);
GeoLine.fVelo:=  REAL_TO_LREAL(NCI_Entry.SyncVelo);
TableDisplayIndex:=  TableDisplayIndex+1;
GeoLine.nDisplayIndex := TableDisplayIndex;
TblPrep.nEntryType:=  GeoLine.nEntryType;
TblPrep.pEntry:=  ADR(GeoLine);
TblPrep.bResetTable:=  FALSE;
END_IF
END_IF
END_ACTION

ACTION M_PTP:
(*Enable, Enable Fw, EnbaleBw这三个 Bit 置 True*)
AxisX.PlcToNc.ControlDWord:=7;
AxisY.PlcToNc.ControlDWord:=7;
(*设置 Override 为 100%, 保留小数点后 4 位的整数*)
AxisX.PlcToNc.Override:=1000000;
AxisX.PlcToNc.Override:=1000000;
END_ACTION

ACTION M_UpdateStatus:
(*设置 Override, 倍率*)
ItpSetOverridePercent(
fOverridePercent := rOverride,
sPlcToNci :=ItpChannel.PlcToNci);
(*获取 GroupI D*)
GroupID := ItpGetGroupId(sNciToPlc:=ItpChannel.NciToPlc );
ChannelID:=ItpGetChannelId(sNciToPlc:=ItpChannel.NciToPlc );
END_ACTION

END_PROGRAM

// ---- POUs/TEST.TcPOU
PROGRAM TEST
VAR
	TEST_STATE1:TEST_STATE;
	j: INT;
END_VAR

CASE TEST_STATE1 OF
	TEST_0:
		j:=10;
		TEST_STATE1:=TEST_1;
	TEST_1:
		j:=j+10;
END_CASE

END_PROGRAM

// ---- POUs/TimeGet.TcPOU
PROGRAM TimeGet
VAR
	NT_GetTime: NT_GetTime;
END_VAR

NT_GetTime(
	NETID:= , 
	START:= , 
	TMOUT:= , 
	BUSY=> , 
	ERR=> , 
	ERRID=> , 
	TIMESTR=> );

END_PROGRAM

// ---- POUs/WAIT.TcPOU
PROGRAM WAIT
VAR
	TON1: TON;
	WAIT_ENABLE: BOOL;
	
	count: INT;
END_VAR


TON1(IN:= TRUE , PT:=T#1MS , Q=> , ET=> );
IF TON1.Q THEN
	TON1(in:= FALSE);
	count := count + 1;
END_IF
//count := count + 1;

END_PROGRAM
